PROGRAM MAIN
VAR
    {attribute 'TcLinkTo' := '.bLimitForwardEnable:=TIIB[Term 2 (EL7031)]^STM Status^Status^Digital input 2;
                              .bLimitBackwardEnable:=TIIB[Term 2 (EL7031)]^STM Status^Status^Digital input 1'}
     M1 : DUT_MotionStage := (nEnableMode:=ENUM_StageEnableMode.ALWAYS, bPowerSelf:=TRUE);
    fbMotionStageM1 : FB_MotionStage;


    {attribute 'pytmc' := '
        pv: SDS:TEST
    '}
    fbCoeReader : FB_Read70x1CoEData;




END_VAR

fbMotionStageM1(stMotionStage:=M1);

fbCoeReader(UserNetId:='172.21.148.67.2.1');

END_PROGRAM

(* stored: Version 1.1.0.1, ProductVersion 3.1.4022.18
   POU MAIN: Id {fb99dda6-98b1-45c2-b37f-6320102b1046}, SpecialFunc None *)
